Omron CX-Programmer project NewProject (CX-Programmer 9.82)

# PLC NewPLC1: CP2E-N N

## Global symbols (name address type ; comment)
0.00 BOOL  ; PB Master On
0.01 BOOL  ; PB EMG
0.02 BOOL  ; Sensor 1
0.03 BOOL  ; Sensor 2
0.04 BOOL  ; Sensor 3
0.05 BOOL  ; Sensor 4
0.06 BOOL  ; Sensor 5
0.07 BOOL  ; Sensor 6
0.08 BOOL  ; Sensor 7
0.09 BOOL  ; Reset
100.00 BOOL  ; Output Sensor 1
100.01 BOOL  ; Output Sensor 1
100.02 BOOL  ; Output Sensor 3
100.03 BOOL  ; Output Sensor 4
100.04 BOOL  ; Output Sensor 5
100.05 BOOL  ; Output Sensor 6
100.06 BOOL  ; Output Sensor 7
3 CHANNEL  ; Timer Detect Product 1
D0 CHANNEL  ; Data Sensor 1
D1 CHANNEL  ; Data Sensor 2
D2 CHANNEL  ; Data Sensor 3
D3 CHANNEL  ; Data Sensor 4
D4 CHANNEL  ; Data Sensor 5
D5 CHANNEL  ; Data Sensor 6
D6 CHANNEL  ; Data Sensor 7
D7 CHANNEL  ; Data Sensor 8

## Program NewProgram1 (cyclic task 0)

### Section Section1

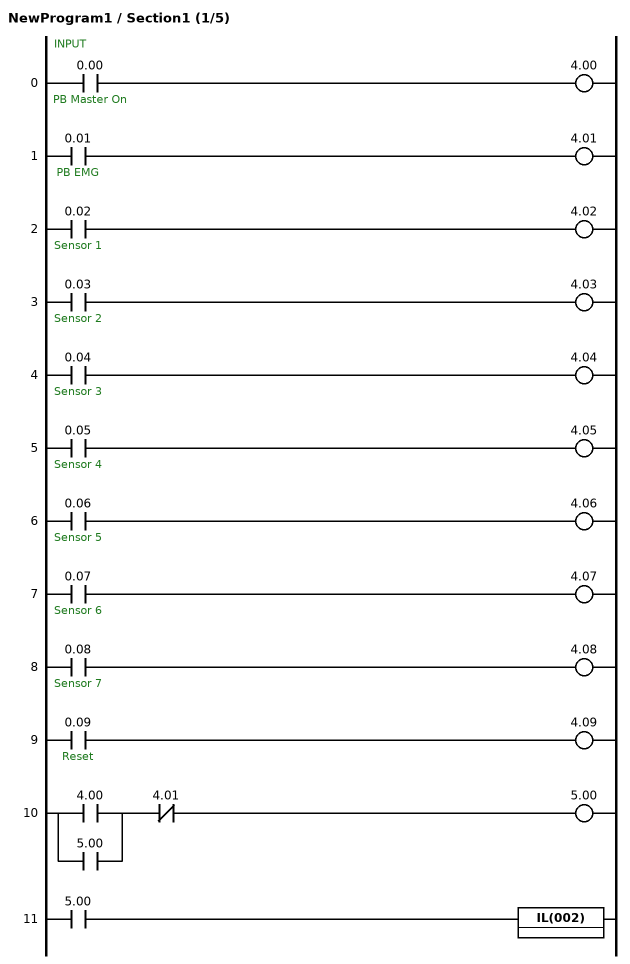
; rung 0: INPUT
LD 0.00  ; PB Master On
OUT 4.00
; rung 1
LD 0.01  ; PB EMG
OUT 4.01
; rung 2
LD 0.02  ; Sensor 1
OUT 4.02
; rung 3
LD 0.03  ; Sensor 2
OUT 4.03
; rung 4
LD 0.04  ; Sensor 3
OUT 4.04
; rung 5
LD 0.05  ; Sensor 4
OUT 4.05
; rung 6
LD 0.06  ; Sensor 5
OUT 4.06
; rung 7
LD 0.07  ; Sensor 6
OUT 4.07
; rung 8
LD 0.08  ; Sensor 7
OUT 4.08
; rung 9
LD 0.09  ; Reset
OUT 4.09
; rung 10
LD 4.00
OR 5.00
ANDNOT 4.01
OUT 5.00
; rung 11
LD 5.00
IL(002)

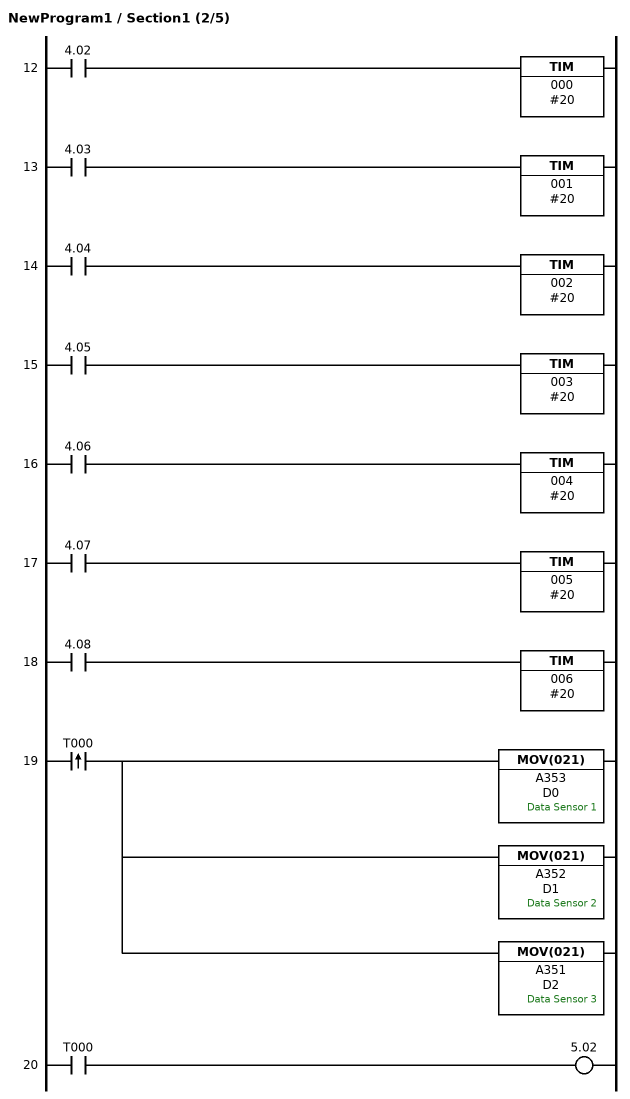
; rung 12
LD 4.02
TIM 000 #20
; rung 13
LD 4.03
TIM 001 #20
; rung 14
LD 4.04
TIM 002 #20
; rung 15
LD 4.05
TIM 003 #20
; rung 16
LD 4.06
TIM 004 #20
; rung 17
LD 4.07
TIM 005 #20
; rung 18
LD 4.08
TIM 006 #20
; rung 19
@LD T000
MOV(021) A353 D0  ; Data Sensor 1
MOV(021) A352 D1  ; Data Sensor 2
MOV(021) A351 D2  ; Data Sensor 3
; rung 20
LD T000
OUT 5.02

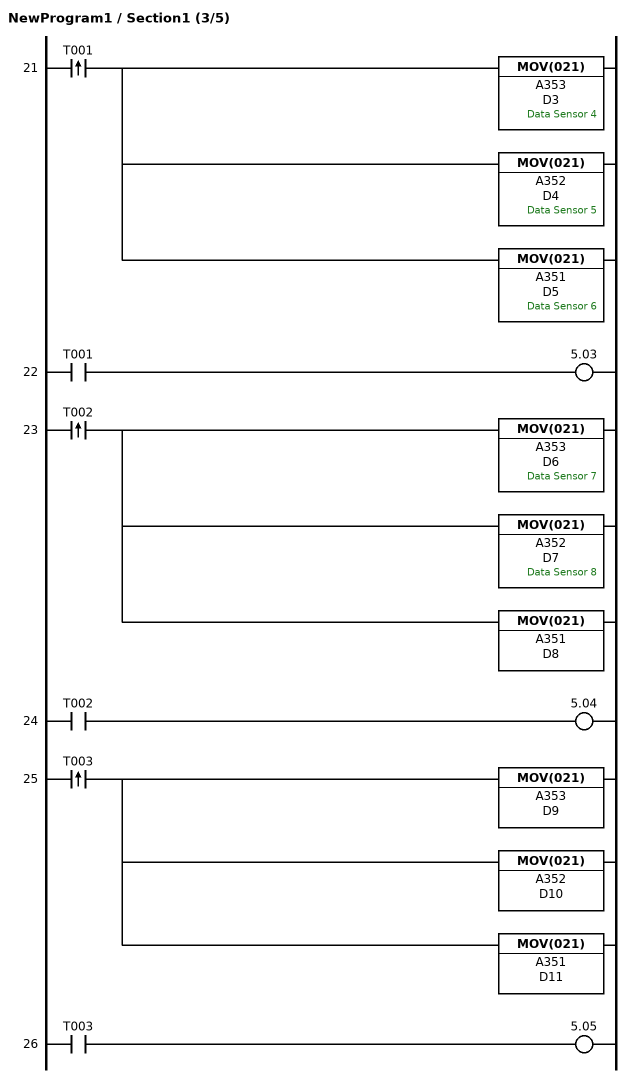
; rung 21
@LD T001
MOV(021) A353 D3  ; Data Sensor 4
MOV(021) A352 D4  ; Data Sensor 5
MOV(021) A351 D5  ; Data Sensor 6
; rung 22
LD T001
OUT 5.03
; rung 23
@LD T002
MOV(021) A353 D6  ; Data Sensor 7
MOV(021) A352 D7  ; Data Sensor 8
MOV(021) A351 D8
; rung 24
LD T002
OUT 5.04
; rung 25
@LD T003
MOV(021) A353 D9
MOV(021) A352 D10
MOV(021) A351 D11
; rung 26
LD T003
OUT 5.05

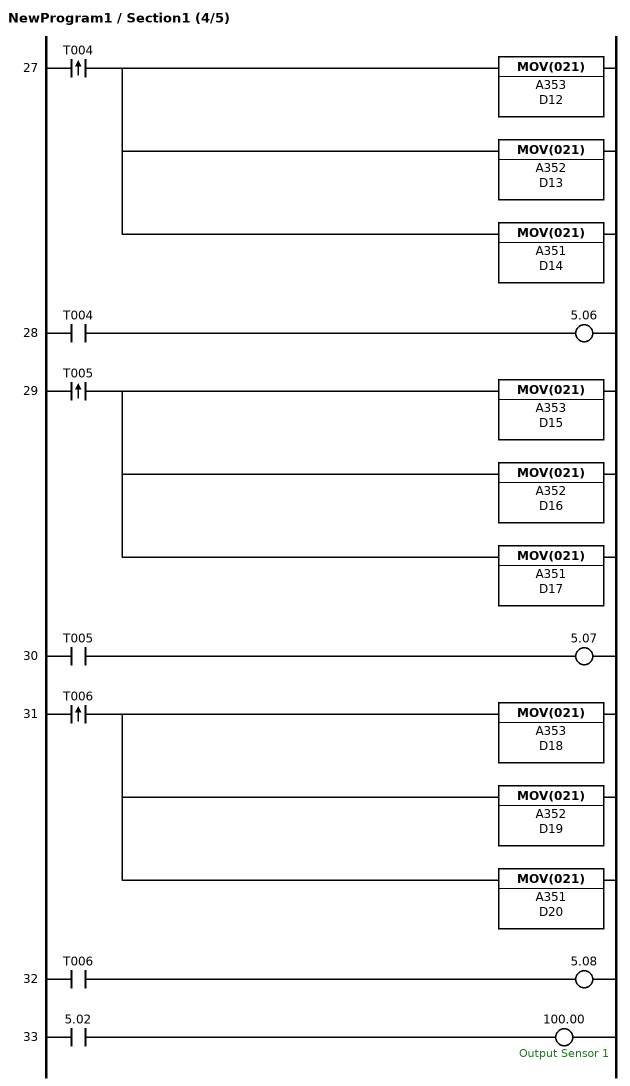
; rung 27
@LD T004
MOV(021) A353 D12
MOV(021) A352 D13
MOV(021) A351 D14
; rung 28
LD T004
OUT 5.06
; rung 29
@LD T005
MOV(021) A353 D15
MOV(021) A352 D16
MOV(021) A351 D17
; rung 30
LD T005
OUT 5.07
; rung 31
@LD T006
MOV(021) A353 D18
MOV(021) A352 D19
MOV(021) A351 D20
; rung 32
LD T006
OUT 5.08
; rung 33
LD 5.02
OUT 100.00  ; Output Sensor 1

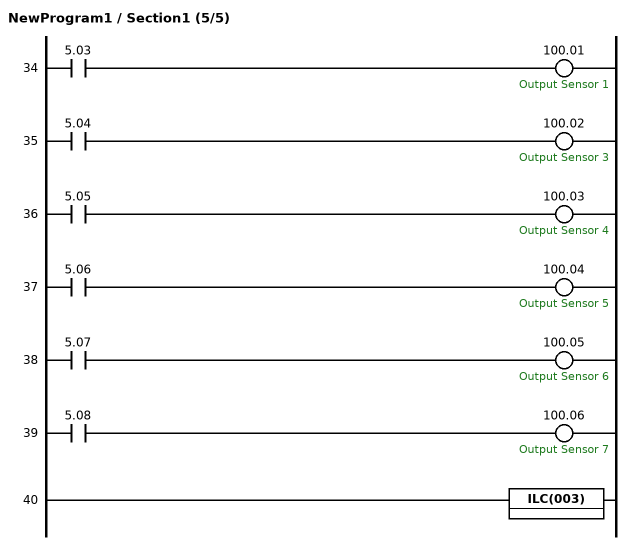
; rung 34
LD 5.03
OUT 100.01  ; Output Sensor 1
; rung 35
LD 5.04
OUT 100.02  ; Output Sensor 3
; rung 36
LD 5.05
OUT 100.03  ; Output Sensor 4
; rung 37
LD 5.06
OUT 100.04  ; Output Sensor 5
; rung 38
LD 5.07
OUT 100.05  ; Output Sensor 6
; rung 39
LD 5.08
OUT 100.06  ; Output Sensor 7
; rung 40
ILC(003)

### Section END
; rung 0
END(001)